FUNCTION_BLOCK FB_Omron_Inv EXTENDS FB_ComponentBase IMPLEMENTS iDM_DriveHealth
VAR
	// Data
	_SetTemperature	   : LREAL;
	_ActualTemperature : LREAL;

	// IO
	_Heat AT %Q* : BOOL;

	// Other items
	RequestedState : eDriveStates	:= eDriveStates.AWAITING_RESET;	
	DriveState : eDriveStates 		:= eDriveStates.FAULT;

	bEnabled : BOOL;
	bInitReversed : BOOL;
	bError : BOOL;
	
	
	eDeviceStatus : eOmronStatus;
	
	bRunningForward : BOOL;
	bRunningReverse : BOOL;
	bFault : BOOL;
	bWarning : BOOL;
	bRemoteEnabled : BOOL;
	bFrequencyMatching : BOOL;
	bConnectionError : BOOL;
	bECDisconnected : BOOL;
	
	blinkErrorAck : FB_BLINKER_PLAY;
	
	tpErrorReset : TP;
	bResetReq : BOOL;
	
	sDriveName : STRING(50);
	tonFailedStartTimeout : TON;
	bResetTried: BOOL;
	
	
//	TempUpdate	 : TON;
//	_InTempRange : BOOL;
END_VAR

ACTION aInputMapping:
bDI1 := stDeviceMapping.inInputTerminal.2;
bDI2 := stDeviceMapping.inInputTerminal.3;
bDI3 := stDeviceMapping.inInputTerminal.4;
bDI4 := stDeviceMapping.inInputTerminal.5;
bDI5 := stDeviceMapping.inInputTerminal.6;
bDI6 := stDeviceMapping.inInputTerminal.0; 
bDI7 := stDeviceMapping.inInputTerminal.1;
bEN1 := stDeviceMapping.inInputTerminal.11;
bEN2 := stDeviceMapping.inInputTerminal.12;


bRunningForward 	:= stDeviceMapping.inStatus.0;
bRunningReverse 	:= stDeviceMapping.inStatus.1;
bFault 				:= stDeviceMapping.inStatus.3;
bWarning 			:= stDeviceMapping.inStatus.7;
bRemoteEnabled		:= stDeviceMapping.inStatus.9;
bFrequencyMatching	:= stDeviceMapping.inStatus.12;
bConnectionError	:= stDeviceMapping.inStatus.15;
bECDisconnected		:= stDeviceMapping.ibWcState;

stDeviceMapping.onFrequencyRef 		:= REAL_TO_UINT(rFreq * 100.0);

bDriveOK := (eDeviceStatus>=4);
bError := eDeviceStatus < eOmronStatus.AWATING_RESET;
END_ACTION

ACTION aSetStatus:
IF bFault AND stDeviceMapping.inSTOActive THEN
	eDeviceStatus := eOmronStatus.AWATING_RESET;
ELSIF bFault THEN
	eDeviceStatus := eOmronStatus.FAULT;
ELSIF bECDisconnected THEN
	eDeviceStatus := eOmronStatus.DRIVE_DISCONNECTED;
ELSIF bConnectionError THEN
	eDeviceStatus := eOmronStatus.CONNECTION_ERROR;
ELSIF bWarning THEN
	eDeviceStatus := eOmronStatus.WARNING;
ELSIF (bRunningForward OR bRunningReverse) AND bFrequencyMatching THEN
	eDeviceStatus := eOmronStatus.RUNNING;
ELSIF bRemoteEnabled THEN
	eDeviceStatus := eOmronStatus.READY;

END_IF
END_ACTION

METHOD PROTECTED CreateEvents
VAR_INPUT
END_VAR
// Add your event creation here
F_CreateAllEventsInClass(Alarms		:= MotionLinxAlarms,
						 ClassSize	:= SIZEOF(TC_EVENTS.MotionlinxAI_Axis),
						 pInitEvent := ADR(TC_EVENTS.MotionlinxAI_Axis.InitReferenceEvent),
						 Prefix		:= Name);

// Super call to base
SUPER^.CreateEvents();
END_METHOD

METHOD CyclicLogic
VAR_INPUT
END_VAR
IF NOT _InitComplete THEN
	_InitComplete := Initialize();
	RETURN;
END_IF

SUPER^.CyclicLogic();

//Read data from Parameters

aInputMapping();
aSetStatus();
END_METHOD

METHOD Disable : BOOL
VAR_INPUT
END_VAR
bEnabled := FALSE;
IF DriveState >= eDriveStates.STOPPED THEN
	RequestedState := eDriveStates.DISABLED;
END_IF
END_METHOD

PROPERTY Drive_State : eDriveStates
GET
Drive_State	:= DriveState;
END_GET
END_PROPERTY

METHOD Enable : BOOL
VAR_INPUT
END_VAR
bEnabled := TRUE;
bResetTried := FALSE;
IF DriveState >= eDriveStates.DISABLED THEN
	RequestedState := eDriveStates.STOPPED;
END_IF
END_METHOD

PROPERTY FaultLocation : STRING(50)
GET
FaultLocation := sDriveName;
END_GET
END_PROPERTY

PROPERTY HasFault : BOOL
GET
HasFault := DriveState = eDriveStates.FAULT;
END_GET
END_PROPERTY

METHOD PROTECTED HMICommunication
VAR_INPUT
END_VAR
SUPER^.HMICommunication();

//Handle the requests to extend and retract
IF ComponentBase_HMI.Status.HMIControlAvailable THEN
	IF MotionlinxAI_HMI.Command.Extend THEN
//		Extend();
	ELSIF MotionlinxAI_HMI.Command.Retract THEN
//		Retract();
	END_IF
END_IF

//Update HMI status info
//Cylinder_HMI.Status.Extended	:= _Extended;
//Cylinder_HMI.Status.Extending	:= _Extending;
//Cylinder_HMI.Status.Retracted	:= _Retracted;
//Cylinder_HMI.Status.Retracting	:= _Retracting;
//Cylinder_HMI.Config.ExtendTime	:= _ExtendTime;
//Cylinder_HMI.Config.RetractTime := _RetractTime;
END_METHOD

PROPERTY IsReady : BOOL
GET
IsReady := DriveState >= eDriveStates.DISABLED;
END_GET
END_PROPERTY

PROPERTY IsRunning : BOOL
GET
IsRunning := bFrequencyMatching;
END_GET
END_PROPERTY

METHOD PROTECTED Monitoring
VAR_INPUT
END_VAR
_Busy	 := IsRunning;
_Error	 := eDeviceStatus < eOmronStatus.AWATING_RESET;
_ErrorID := ;//eError;
SUPER^.Monitoring();
END_METHOD

PROPERTY STO_Active : bool
GET
END_GET
END_PROPERTY

END_FUNCTION_BLOCK

(* stored: Version 1.1.0.1, ProductVersion 3.1.4024.16
   POU FB_Omron_Inv: Id {1f5cda4b-8c9e-495c-9cbf-e32b31d9573a}, SpecialFunc None
   Folder I_ComponentBase: Id {036e2951-221f-432b-806a-55d1520966ba}
   Folder I_CyclicFB: Id {0ba0ab25-9c32-4537-8f9a-d985458c36e5}
   Folder I_Omron_Axis: Id {c82a40de-4317-48a4-aebf-f7596bbe1a82}
   Action aInputMapping: Id {71f983bd-d03d-48e8-8561-3f3c3aed0abd}
   Action aSetStatus: Id {5e1d199c-9d3f-42a0-af71-fea74cffbb68}
   Method CreateEvents: Id {102abde3-039c-4fb2-9376-991a4a0807d0}
   Method CyclicLogic: Id {347c823a-8712-4a6c-978f-6cf5d5a172b0}
   Method Disable: Id {51733576-a092-440d-a7bd-6868f4006402}
   Property Drive_State: Id {180f5dad-82e1-498b-8484-b720740bbc42}
   Get Get: Id {f04b2a6b-f072-4177-91be-c6b7079b22f7}
   Method Enable: Id {28b8211c-4512-40a4-9c99-144320355d2f}
   Property FaultLocation: Id {2fee8a38-4fea-47c1-8e0c-94be448d8c3c}
   Get Get: Id {2c1d3040-21b2-4b31-9e69-c1c39684a509}
   Property HasFault: Id {e20fc962-7a91-45ca-ac92-c5c86d30c2c2}
   Get Get: Id {033e052a-64b0-4857-bb09-d0357140eb4d}
   Method HMICommunication: Id {8f26cd40-35db-4ae2-818a-c456dc6440b9}
   Property IsReady: Id {780811cb-7987-44e6-bc08-d56d0f1608ac}
   Get Get: Id {48a107da-0acc-46f5-9f1f-7bf2b2ed5bb5}
   Property IsRunning: Id {dce4b26a-f544-47e1-b4f0-3170eb436490}
   Get Get: Id {3c7fb4f9-31ed-4043-8822-5d201a37ae38}
   Method Monitoring: Id {6476d871-905c-47fc-9c3f-e47c04830768}
   Property STO_Active: Id {8d1988dc-7175-47f5-9aee-b8aa192860e1}
   Get Get: Id {3d088828-3760-43e6-b798-72f24a666139} *)
